FUNCTION_BLOCK ASTORAGE_DEMUX (* Composite FB wrapping other FBs *)
  (* Standard: 61499-2 *)
  (* Version 0.0, 2008-07-10, 4DIAC-IDE, 4DIAC-Consortium *)
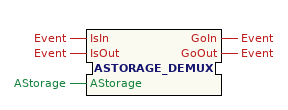
  EVENT_INPUT
    IsIn; (* Request from Socket *)
    IsOut; (* Response from Socket *)
  END_EVENT
  EVENT_OUTPUT
    GoIn; (* Confirmation from Plug *)
    GoOut;
  END_EVENT
  SOCKETS
    AStorage : AStorage;
  END_SOCKETS
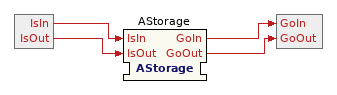
  EVENT_CONNECTIONS
    IsIn TO AStorage.IsIn;
    IsOut TO AStorage.IsOut;
    AStorage.GoIn TO GoIn;
    AStorage.GoOut TO GoOut;
  END_CONNECTIONS
END_FUNCTION_BLOCK
